{attribute 'GeneratedUsingTerminal: KL2532'}
{attribute addProperty BoxType "KL2532"}
{attribute addProperty Id "StateAT %I*USINT0Data_InAT %I*INT0CtrlAT %Q*USINT0Data_OutAT %Q*INT0"}
{attribute addProperty CRC "1702274689"}
{attribute addProperty Size "0"}
TYPE Channel_6576A681 :
STRUCT
	{attribute addProperty Name "State"}
	State AT %I* : USINT;
	{attribute addProperty Name "Data_In"}
	Data_In AT %I* : INT;
	{attribute addProperty Name "Ctrl"}
	Ctrl AT %Q* : USINT;
	{attribute addProperty Name "Data_Out"}
	Data_Out AT %Q* : INT;
END_STRUCT
END_TYPE

(* stored: Version 1.2.0.0, ProductVersion 3.1.4024.11
   DUT Channel_6576A681: Id {8641fad8-4af0-4f5d-9237-07b3b3629d7d} *)
